FUNCTION_BLOCK FB_FeedforwardWinch
VAR_INPUT
	bEnable		: BOOL;
	fInput_ms	: LREAL;
	fDisplacment_cc : LREAL;
	rCircumference : REAL;
	stOpenLoopControlSettings : ST_OpenLoopControlSettings;
	rTransmission : REAL;
END_VAR
VAR_OUTPUT
	fNormalizedOutput: LREAL;
END_VAR
VAR
	fFlowReference_lmin : LREAL;
	fRads : LREAL;
END_VAR

fRads := fInput_ms * 3.14 * 2 * rTransmission / (rCircumference);
fFlowReference_lmin := (fDisplacment_cc*1E-5*fRads/(2*3.14))*60000;

IF bEnable THEN 
    fNormalizedOutput := (fFlowReference_lmin) / stOpenLoopControlSettings.fMaxFlowCapacity;
ELSE 
    fNormalizedOutput := 0.0;
END_IF;

IF fNormalizedOutput > 1.0 THEN
    fNormalizedOutput := 1.0;
ELSIF fNormalizedOutput < -1.0 THEN 
    fNormalizedOutput := -1.0;
END_IF;

END_FUNCTION_BLOCK

(* stored: Version 1.1.0.1, ProductVersion 3.1.4024.11
   POU FB_FeedforwardWinch: Id {33c27b48-71a3-4f77-967b-ab3f6d50d321}, SpecialFunc None *)
